VAR_GLOBAL

	EX_LoadCell	: fbHBMSerialCtrl;
	EX_LoadCellVar:	structHBMSerialCtrl;	

END_VAR

(* stored: Version 1.1.0.1, ProductVersion 3.1.4018.2
   GVL GVL_LoadCell: Id {56592926-0278-4d03-ad64-2d5eb601d62e} *)
